TYPE McReadBoolParameterArgs :
STRUCT
	///Number of the parameter
	parameterNumber: INT;
END_STRUCT
END_TYPE

(* stored: Version 1.1.0.1, ProductVersion 3.1.4019.2
   DUT McReadBoolParameterArgs: Id {9264d4d4-2db4-407c-8eb1-39adcc78cba6} *)
